Staubli VAL3: SimpleMessage.dtx

public _CommType CommType
  [0]
    num INVALID
    num SERVICE_REPLY
    num SERVICE_REQUEST
    num TOPIC
public _MsgType MsgType
  [0]
    num GET_VERSION
    num JOINT_FEEDBACK
    num JOINT_POSITION
    num JOINT_TRAJ
    num JOINT_TRAJ_PT
    num JOINT_TRAJ_PT_F
    num PING
    num STATUS
public _ReplyCode ReplyCode
  [0]
    num FAILURE
    num INVALID
    num SUCCESS
public _SpecialSeqVal SpecialSeqVal
  [0]
    num END_TRAJECTORY
    num START_TRAJ_DOWN
    num START_TRAJ_STRE
    num STOP_TRAJECTORY
